# EPICS substitutions: hp8xxxaApp/Db/hp8xxxa.substitutions
file hp8xxxaCh.template{
    {N=1}
    {N=4}
}
file hp8xxxaCtrl.db{
    {N=0}
}
